FUNCTION_BLOCK EventLogger
VAR
	EventBuffer : ARRAY[1..EVENT_BUFFER_MAX_SIZE] OF ST_Event;
	CurrentEventBufferIndex : INT := 0;
	_PersistentEventStorage : I_PersistentEventStorage;
END_VAR
VAR CONSTANT
	EVENT_BUFFER_MAX_SIZE : INT := 100;
END_VAR

METHOD PUBLIC AddEvent : BOOL
VAR_INPUT
	eEventType : E_EventType;
	eEventSeverity : TcEventSeverity;
	nEventIdentity : UDINT;
	sEventText : STRING(255);
END_VAR
IF NOT IsEventBufferFull() THEN
	//todo
	CurrentEventBufferIndex := CurrentEventBufferIndex + 1;
	EventBuffer[CurrentEventBufferIndex].eEventType := eEventType;
	EventBuffer[CurrentEventBufferIndex].eEventSeverity := eEventSeverity;
	EventBuffer[CurrentEventBufferIndex].nEventIdentity := nEventIdentity;
	EventBuffer[CurrentEventBufferIndex].sEventText := sEventText;
	F_UpdateEventTimestampWithSystemTime(stEvent := EventBuffer[CurrentEventBufferIndex]); 
	AddEvent := TRUE;
ELSE
	AddEvent := FALSE;
END_IF

_PersistentEventStorage.StoreEvent(stEvent := EventBuffer[CurrentEventBufferIndex]);
END_METHOD

METHOD FB_Init : BOOL
VAR_INPUT
	bInitRetains : BOOL;
	bInCopyCode : BOOL;
	iPersistentEventStorage : I_PersistentEventStorage;
END_VAR
_PersistentEventStorage := iPersistentEventStorage;
END_METHOD

METHOD PRIVATE IsEventBufferFull : BOOL
IF (CurrentEventBufferIndex + 1) >= EVENT_BUFFER_MAX_SIZE THEN
	IsEventBufferFull := TRUE;
ELSE
	IsEventBufferFull := FALSE;
END_IF
END_METHOD

METHOD print1 : BOOL
VAR_INPUT
	level : TcEventSeverity;
	str1 : STRING;
END_VAR

VAR
	enum_as_text : STRING;
END_VAR
CASE level OF
	TcEventSeverity.Critical:
		enum_as_text := '[CRITICAL] ';
	TcEventSeverity.Error:
		enum_as_text := '[ERROR] ';
	TcEventSeverity.Warning:
		enum_as_text := '[WARNING] ';		
	TcEventSeverity.Info:
		enum_as_text := '        [INFO] ';
	TcEventSeverity.Verbose:
		enum_as_text := '                        [VERBOSE] ';
END_CASE

IF (TO_SINT(level) >= MAIN.minimumLogSeverity) THEN
	ADSLOGSTR(ADSLOG_MSGTYPE_ERROR, 
              CONCAT(enum_as_text, str1), 
              '');
END_IF
END_METHOD

METHOD print2 : BOOL
VAR_INPUT
	level : TcEventSeverity;
	str1 : STRING;
	str2 : STRING;
END_VAR

VAR
	enum_as_text : STRING;
END_VAR
CASE level OF
	TcEventSeverity.Critical:
		enum_as_text := '[CRITICAL] ';
	TcEventSeverity.Error:
		enum_as_text := '[ERROR] ';
	TcEventSeverity.Warning:
		enum_as_text := '[WARNING] ';		
	TcEventSeverity.Info:
		enum_as_text := '        [INFO] ';
	TcEventSeverity.Verbose:
		enum_as_text := '                        [VERBOSE] ';
END_CASE

IF (TO_SINT(level) >= MAIN.minimumLogSeverity) THEN
	ADSLOGSTR(ADSLOG_MSGTYPE_ERROR, 
			  CONCAT(enum_as_text, str1), 
			  str2);
END_IF
END_METHOD

END_FUNCTION_BLOCK

(* stored: Version 1.1.0.1, ProductVersion 3.1.4024.12
   POU EventLogger: Id {49a270de-7b38-4c0a-b542-93db06ca3178}, SpecialFunc None
   Folder logging: Id {863f0790-67e2-4cc6-8b30-85c6b211446d}
   Method AddEvent: Id {8442e16c-f730-4c65-b703-9df028836144}
   Method FB_Init: Id {732d1647-b707-4d0e-b915-0e3d09f67b76}
   Method IsEventBufferFull: Id {6c0e3054-2059-437d-ace7-75813699a690}
   Method print1: Id {7f43a41b-9e98-4aa2-a748-dcf5656a0706}
   Method print2: Id {287da7bd-5655-405b-bd79-4e59ca6d7cd7} *)
